FUNCTION_BLOCK SawmillSpeed
  (* Standard: 61499-2 *)
  (* Version 0.1, 2017-00-27, Hammond, HAMMONDSDESKTOP *)
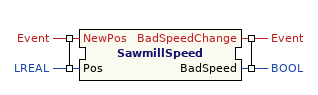
  EVENT_INPUT
    NewPos WITH Pos;
  END_EVENT
  EVENT_OUTPUT
    BadSpeedChange WITH BadSpeed;
  END_EVENT
  VAR_INPUT
    Pos : LREAL;
  END_VAR
  VAR_OUTPUT
    BadSpeed : BOOL;
  END_VAR
  VAR
    LastPos : LREAL;
  END_VAR
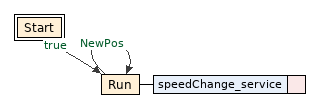
  EC_STATES
    Start;
    Run : speedChange_service;
  END_STATES
  EC_TRANSITIONS
    Start TO Run := true;
    Run TO Run := NewPos;
  END_TRANSITIONS
  ALGORITHM speedChange_service IN C:
if(me->LastPos != 0) {
	if(me->NewPos - me->LastPos > 2 || me->LastPos - me->NewPos > 2) {
		me->outputEvents.event.BadSpeedChange = 1;
		me->BadSpeed = true;
	} else {
		me->outputEvents.event.BadSpeedChange = 1;
		me->BadSpeed = false;
	}
}

me->LastPos = me->NewPos;
  END_ALGORITHM
END_FUNCTION_BLOCK
